FUNCTION_BLOCK E_TONOF (* standard timer function block (on/off-delay timing) *)
  (* Standard: 61499-2; Classification: standard timer function block; Description: Copyright (c) 2024 HR Agrartechnik GmbH This program and the accompanying materials are made available under the terms of the Eclipse Public License 2.0 which is available at https://www.eclipse.org/legal/epl-2.0/ SPDX-License-Identifier: EPL-2.0 E_TONOF -- On/Off-delay timer FB When IN goes TRUE, Q becomes TRUE after delay PT_ON. When IN goes FALSE, Q becomes FALSE after delay PT_OFF. Reset stops both timers and sets Q to FALSE. *)
  (* Version 3.1, 2026-05-08, Franz Höpfinger, HR Agrartechnik GmbH, E_RF_TRIG instead of E_SWITCH *)
  (* Version 3.0, 2025-04-14, Patrick Aigner, changed package *)
  (* Version 1.1, 2024-04-23, Franz Höpfinger, HR Agrartechnik GmbH, Add a Reset to Timer FBs *)
  (* Version 1.0, 2024-03-04, Franz Höpfinger, HR Agrartechnik GmbH *)
  PACKAGE iec61499::events::timers;
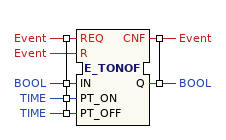
  EVENT_INPUT
    REQ WITH IN, PT_ON, PT_OFF; (* Normal Execution Request *)
    R; (* Reset *)
  END_EVENT
  EVENT_OUTPUT
    CNF WITH Q; (* Execution Confirmation *)
  END_EVENT
  VAR_INPUT
    IN : BOOL; (* Input *)
    PT_ON : TIME; (* Process time ON Delay *)
    PT_OFF : TIME; (* Process time OFF Delay *)
  END_VAR
  VAR_OUTPUT
    Q : BOOL; (* Output *)
  END_VAR
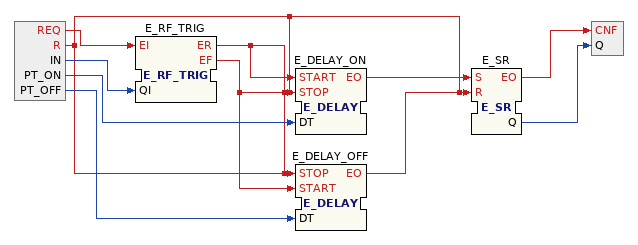
  FBS
    E_RF_TRIG : iec61499::events::E_RF_TRIG;
    E_DELAY_ON : iec61499::events::E_DELAY;
    E_SR : iec61499::events::E_SR;
    E_DELAY_OFF : iec61499::events::E_DELAY;
  END_FBS
  EVENT_CONNECTIONS
    REQ TO E_RF_TRIG.EI;
    E_DELAY_ON.EO TO E_SR.S;
    E_SR.EO TO CNF;
    E_DELAY_OFF.EO TO E_SR.R;
    R TO E_SR.R;
    R TO E_DELAY_OFF.STOP;
    E_RF_TRIG.ER TO E_DELAY_ON.START;
    E_RF_TRIG.EF TO E_DELAY_ON.STOP;
    E_RF_TRIG.ER TO E_DELAY_OFF.STOP;
    E_RF_TRIG.EF TO E_DELAY_OFF.START;
    R TO E_DELAY_ON.STOP;
  END_CONNECTIONS
  DATA_CONNECTIONS
    IN TO E_RF_TRIG.QI;
    PT_ON TO E_DELAY_ON.DT;
    E_SR.Q TO Q;
    PT_OFF TO E_DELAY_OFF.DT;
  END_CONNECTIONS
END_FUNCTION_BLOCK
